Staubli VAL3: commandCheck.pgx

program commandCheck(num& nArgs[] (dimensions=1), num nNbArgs (dimensions=1), string& sBuffer (dimensions=1), string sCommand (dimensions=1), bool& bFlag (dimensions=1))
begin
  //check command name and arguments
  //everything passed by reference from serverCmd
  bFlag=false
  //popUpMsg(sCommand)
  switch sCommand
    case "gripper"
      if nNbArgs!=1
        sBuffer="NACK: "+sCommand+" nNbArgs: "+chr(nNbArgs)
      else
        if (nArgs[0]<0) or (nArgs[0]>1)
          sBuffer="NACK: "+sCommand+" nArgs[0]: "+chr(nArgs[0])
        else
          bFlag=true
        endIf
      endIf
    break
    case "pickTool"
      if nNbArgs!=1
        sBuffer="NACK: "+sCommand+" nNbArgs: "+chr(nNbArgs)
      else
        if (nArgs[0]<0) or (nArgs[0]>1)
          sBuffer="NACK: "+sCommand+" nArgs[0]: "+chr(nArgs[0])
        else
          bFlag=true
        endIf
      endIf
    break
    case "power"
      if nNbArgs!=1
        sBuffer="NACK: "+sCommand+" nNbArgs: "+toString("",nNbArgs)
      else
        if (nArgs[0]<0) or (nArgs[0]>1)
          sBuffer="NACK: "+sCommand+" nArgs[0]: "+toString("",nArgs[0])
        else
          bFlag=true
        endIf
      endIf
    break
    case "stopMove"
      if nNbArgs!=0
        sBuffer="NACK: "+sCommand+" nNbArgs: "+chr(nNbArgs)
      else
        bFlag=true
      endIf
    break
    case "restartMove"
      if nNbArgs!=0
        sBuffer="NACK: "+sCommand+" nNbArgs: "+chr(nNbArgs)
      else
        bFlag=true
      endIf
    break
    case "deleteMove"
      if nNbArgs!=0
        sBuffer="NACK: "+sCommand+" nNbArgs: "+chr(nNbArgs)
      else
        bFlag=true
      endIf
    break
    case "isSettled"
      if nNbArgs!=0
        sBuffer="NACK: "+sCommand+" nNbArgs: "+chr(nNbArgs)
      else
        bFlag=true
      endIf
    break
    case "setFrame"
      if nNbArgs!=1
        sBuffer="NACK: "+sCommand+" nNbArgs: "+chr(nNbArgs)
      else
        if (nArgs[0]<0) or (nArgs[0]>3)
          sBuffer="NACK: "+sCommand+" nArgs[0]: "+chr(nArgs[0])
        else
          bFlag=true
        endIf
      endIf
    break
    case "setTool"
      if nNbArgs!=1
        sBuffer="NACK: "+sCommand+" nNbArgs: "+chr(nNbArgs)
      else
        if (nArgs[0]<0) or (nArgs[0]>3)
          sBuffer="NACK: "+sCommand+" nArgs[0]: "+chr(nArgs[0])
        else
          bFlag=true
        endIf
      endIf
    break
    case "moveX"
      if nNbArgs!=1
        sBuffer="NACK: "+sCommand+" nNbArgs: "+chr(nNbArgs)
      else
        if abs(nArgs[0])>50
          sBuffer="NACK: "+sCommand+" nArgs[0]: "+chr(nArgs[0])
        else
          bFlag=true
        endIf
      endIf
    break
    case "moveY"
      if nNbArgs!=1
        sBuffer="NACK: "+sCommand+" nNbArgs: "+chr(nNbArgs)
      else
        if abs(nArgs[0])>50
          sBuffer="NACK: "+sCommand+" nArgs[0]: "+chr(nArgs[0])
        else
          bFlag=true
        endIf
      endIf
    break
    case "moveZ"
      if nNbArgs!=1
        sBuffer="NACK: "+sCommand+" nNbArgs: "+chr(nNbArgs)
      else
        if abs(nArgs[0])>50
          sBuffer="NACK: "+sCommand+" nArgs[0]: "+chr(nArgs[0])
        else
          bFlag=true
        endIf
      endIf
    break
    case "getX"
      if nNbArgs!=0
        sBuffer="NACK: "+sCommand+" nNbArgs: "+chr(nNbArgs)
      else
        bFlag=true
      endIf
    break
    case "getY"
      if nNbArgs!=0
        sBuffer="NACK: "+sCommand+" nNbArgs: "+chr(nNbArgs)
      else
        bFlag=true
      endIf
    break
    case "getZ"
      if nNbArgs!=0
        sBuffer="NACK: "+sCommand+" nNbArgs: "+chr(nNbArgs)
      else
        bFlag=true
      endIf
    break
    default
      logMsg("commandCheck fail: "+sCommand)
    break
  endSwitch
  //
end
